// TIA Portal V16 export
// export: Created 2021-04-06T19:52:17.511393Z, ExportSetting WithDefaults, DisplayName Totally Integrated Automation Portal, DisplayVersion V16, DisplayName TIA Portal Version Control Interface, DisplayVersion V16, DisplayName TIA Portal Openness, DisplayVersion V16, DisplayName STEP 7 Professional, DisplayVersion V16, DisplayName STEP 7 Safety, DisplayVersion V16, DisplayName WinCC Unified SCADA Engineering System, DisplayVersion V16
FUNCTION_BLOCK "Sorting_AM"   // FB13, LAD
TITLE = Блок сортировки
{ S7_Optimized_Access := 'TRUE' }
VERSION : 0.1
// Из массива ReadyToSort считываем количество заполненых бункеров. Если их больше либо равно 6 то начинаем сортировку.
// После нахождения искомых бункеров формируем массив readyToDrop.
// После путем перемножения ReadyToSort *Not(readyToDrop) исключаем сбрасывемые бункера из сортировки
// stored: AutoNumber true, IsIECCheckEnabled false, IsRetainMemResEnabled false, MemoryReserve 100, SetENOAutomatically false, UDAEnableTagReadback false
   VAR_INPUT
      enableToWork : Bool;   // разрешение на работу блока
      setWeight : Real;   // итоговый разыскиваемый вес
      errorMeasurement : Real;   // погрешность
      isWorkWithBunker : Array[0..12] of Bool;   // разрешение работать с конкретными бункерами
      setWeightBunker { ExternalAccessible := 'False'; ExternalVisible := 'False'; ExternalWritable := 'False'} : Array[0..12] of Real;   // уставки весов в бункерах
   END_VAR
   VAR_IN_OUT
      stableWeightBunker : Array[0..12] of Real;   // стабильный вес в бункерах
      readyToSorting : Array[0..12] of Bool;   // готовность бункеров к сортировке
      readyToDrop : Array[0..12] of Bool;   // итоговый сигнал сортировки для сброса на конвейер
      blockSort : Bool;   // блокировать сортировку чтобы просто скинуть все готовые
   END_VAR
   VAR
      valueReadyToDrop { ExternalAccessible := 'False'; ExternalVisible := 'False'; ExternalWritable := 'False'} : Bool;
      valueReadytoSortBunker : SInt;   // количество бункеров готовых к сортировке
      valueIsWorkWithBunker : SInt;
      tmpStableWeight : Array[0..12] of Real;   // массив с весами которые будем сортировать
      bufferReadyToDrop : Array[0..12] of Bool;   // на случай того что если readyToDrop не был сброшен
      Sort_Real_FB : "Sort_Real";
      full1 : Array[0..12] of Bool;
      full0 : Array[0..12] of Bool;
   END_VAR
   VAR_TEMP
      i : SInt;
      j : SInt;
      k : SInt;
      l : SInt;
      "m" : SInt;
      tmpReadyToDrop : Array[0..12] of Bool;   // временный массив готовности к сбросу
      minWeight : Real;
      tmpArrayBlock : Array[0..12] of Bool;   // временный массив на проверку все ли бункера готовы при блокировке
      tmpArrNotDrop : Array[0..12] of Real;
      tmpSumFind : Real;
      indexTmpSumFind : SInt;
      noDrop : SInt;
      stateFindIndex : Bool;
   END_VAR
   // full1[1..12] := true;
BEGIN

REGION Network 1 (SCL): Определяем ValueToSortBunker
   IF #enableToWork THEN //разрешение на работу блока 
       //необходимо проверить не подготовил ли блок сортировки уже значения для сброса
       #valueReadyToDrop := false;
       #i := 0;
       FOR #i := 1 TO 12 DO
           IF #readyToDrop[#i] THEN
               #valueReadyToDrop := true;
               EXIT;//выходим из FOR тк то что надо уже нашли
           END_IF;
       END_FOR;

       IF NOT (#valueReadyToDrop) THEN
           //если сортировку не производили
           #i := 0;
           #valueIsWorkWithBunker := 0;
           #valueReadytoSortBunker := 0;
           FOR #i := 1 TO 12 DO
               //подсчитаем количесво бункеров с которыми можно работать
               //и какие готовы к сортировке
               //
               IF #isWorkWithBunker[#i] THEN
                   #valueIsWorkWithBunker := #valueIsWorkWithBunker + 1;
               END_IF;
               IF #readyToSorting[#i] = #isWorkWithBunker[#i] THEN
                   #valueReadytoSortBunker := #valueReadytoSortBunker + 1;
               END_IF;
           END_FOR;

           IF #blockSort THEN
               //если включена блокировка то просто ждем готовности бункеров к сортировке
               //
               IF #valueIsWorkWithBunker = #valueReadytoSortBunker THEN
                   //если число готовых к сортировке бункеров совпадает 
                   //с числом разрешенных к работе в режиме блокировки то
                   //просто скидываем все
                   #tmpReadyToDrop := #readyToSorting;
               END_IF;
           ELSE
               //если блокировки нет то сортируем по стандарту

               // IF #valueIsWorkWithBunker = 1 THEN
               //     //если бункеров разрешенных к работе один то 
               //     #i := 0;
               //     FOR #i := 1 TO 12 DO //заполняем временный массив готовности к сбросу
               //         #tmpReadyToDrop[#i] := #readyToSorting[#i] AND #isWorkWithBunker[#i];
               //     END_FOR;
               // ELSE

               IF #valueReadytoSortBunker >= 5 THEN//начинаем сортировку
                   #i := 0;
                   FOR #i := 1 TO 12 DO//определим массив чисел с которыми будем работать
                       #tmpStableWeight[#i] := #stableWeightBunker[#i] * BOOL_TO_INT(#readyToSorting[#i]);
                   END_FOR;
                   //далее работаем только с весами из массива #tmpStableWeight
                   //

                   //*****************************
                   //временная заглушка - скидываем бункера которые тупа в сумме
                   //дают больше либо равно уставке
                   //
                   #tmpArrNotDrop := #tmpStableWeight;

                   //#Sort_Real_FB(array := #tmpArrNotDrop);
                   //теперь массив #tmpArrNotDrop отсортирован и числа которые 
                   //мы можем использовать начинаются с индекса (12-noDrop+1)
                   #k := 0;
                   #tmpSumFind := 0;//где храним сумму
                   #stateFindIndex := false;
                   #indexTmpSumFind := 0;//индекс элемента массива на котором надо остановиться
                   //#noDrop := #valueReadytoSortBunker;
                   FOR #k := 1 TO 12 DO
                       #tmpSumFind := #tmpSumFind + #tmpArrNotDrop[#k];
                       IF #tmpSumFind >= #setWeight//если попадаем 
                       THEN
                           #stateFindIndex := true;
                           #indexTmpSumFind := #k;
                           EXIT;//выходим из FOR
                       END_IF;

                   END_FOR;
                   IF NOT (#stateFindIndex) THEN //ничего не нашли
                       #tmpReadyToDrop := #full0;
                   ELSE
                       #l := 0;//заполняем массив на сброс
                       FOR #l := 1 TO #indexTmpSumFind DO
                           IF #tmpArrNotDrop[#l] > 0 THEN
                               #tmpReadyToDrop[#l] := true;
                           END_IF;
                       END_FOR;

                   END_IF;
                   //*************************************


                   //корректируем массив readyToSorting
                   #i := 0;
                   FOR #i:= 1 TO 12 DO
                       IF #tmpReadyToDrop[#i] THEN
                           #readyToSorting[#i] := false;
                       END_IF;
                   END_FOR;
               END_IF;
           END_IF;
       ELSE
           #tmpReadyToDrop := #readyToDrop;//если значения уже были
           //и не сброшены то сортировку не производили
       END_IF;

   END_IF;



   #readyToDrop := #tmpReadyToDrop;//переписываем из временного в блочный
END_REGION
END_FUNCTION_BLOCK
